(* PLC project Unnamed, Unknown Unnamed 1 *)
(* stored: creationDateTime 2021-08-22T15:13:27, modificationDateTime 2021-08-22T15:38:24 *)

PROGRAM program1
  VAR
    x : BOOL;
    y : BOOL;
    z : BOOL;
  END_VAR

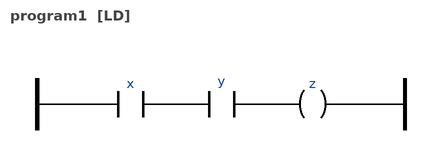
(* LD diagram, written out as Structured Text *)
z := x AND y;
END_PROGRAM

CONFIGURATION Config0
  RESOURCE Res0 ON PLC
    TASK task0(INTERVAL := T#20ms, PRIORITY := 0);
    PROGRAM instance0 WITH task0 : program1;
  END_RESOURCE
END_CONFIGURATION
